# EPICS substitutions: ps300Sup/devSRS_PS370.substitutions
##########################################################################
# Copyright (c) 2012 Lawrence Berkeley National Laboratory, Accelerator
# Technology Group, Engineering Division
# This code is distributed subject to a Software License Agreement found
# in file LICENSE that is included with this distribution.
##########################################################################

file devSRS_PS3xx.template
{
  { P="\$(P)", R="\$(R)", PORT="\$(PORT)", A="\$(A)",
  VMIN="-20000", VMAX="-100", IMIN="0", IMAX="525e-6" }
}
